Fanuc KAREL source: ks00056.KL

-- PROVISIONAL review KL for V770-1; original PC SHA256 b1798b20bd42ce844f2008b871b6d8a39573d2469ef180f6f1a45bf87b8d6fd5
-- Incomplete behavior may be omitted. Consult companion uncertainty JSON. Do not deploy.
PROGRAM KS00056
%NOLOCKGROUP
BEGIN
  -- UNRESOLVED_PC offsets 5-13; opcodes 3F,75
  -- UNRESOLVED_PC offsets 18-27; opcodes 3F,75
  -- UNRESOLVED_PC offsets 32-70; opcodes 27,22,22,2A,22,2A,22,22,B0
  -- UNRESOLVED_PC offsets 75-79; opcodes 7F
END KS00056
